VAR_GLOBAL
    // Achsen ***************************************************	
	X_Achse_steuern						: DUT_Achse_Steuern;	
	X_Achse_status						: DUT_Achse_Status;	
		                            	
	Y_Achse_steuern						: DUT_Achse_Steuern;		
	Y_Achse_status						: DUT_Achse_Status;		
	
	Z_Achse_steuern						: DUT_Achse_Steuern;			
	Z_Achse_status						: DUT_Achse_Status;		

    // Frequenzumrichter ****************************************
	Bohraggr_Stufenbohr_steuern			: DUT_SEW_FU_Steuern;	
	Bohraggr_Stufenbohr_status			: DUT_SEW_FU_Status;
	Bohraggr_Stulpfraes_steuern			: DUT_SEW_FU_Steuern;	
	Bohraggr_Stulpfraes_status			: DUT_SEW_FU_Status;

    // Ventile **************************************************
    Vorbohren_Bohrhub          			: DUT_Ventil_sps;
    Stulpfraes_Vorlegehub      			: DUT_Ventil_sps;
    Pusher				             	: DUT_Ventil_sps;
    Schienenklemm		             	: DUT_Ventil_sps;

    // interne Variablen ****************************************
    sk_Freigabe                         : BOOL;
    sk                                  : INT;
    transport_einfoerdern_bereit        : BOOL;
    transport_ausfoerdern_bereit        : BOOL;

    Tuer_Anwahl                         : BOOL;   // Signal Tür Anwahl, Tür soll geöffnet werden
    Tuer_Freigabe                       : BOOL;   // Signal Tür Freigabe, Tür kann geöffnet werden
END_VAR

(* stored: Version 1.1.0.1
   GVL GVL_3200: Id {3633ca40-8307-4abc-ad17-2687e22ce9a1} *)
